# B&R Automation Studio project Myjnia
Automation Studio 4.9.3.144 SP; technology packages: mappView 5.12.1

## Configuration Config1

CPU X20CP1382, AutomationRuntime B4.83, Build 4.1.2, Vc V4.72.2

### Task classes (Cpu.sw)
```
Cyclic#4:
  Program <- Program.prg
VcDataObjects: Visu <- Visu.dob
```

### Hardware
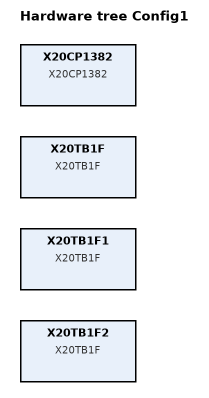
```
X20CP1382 : X20CP1382 v1.11.0.0  [X1 -> X1.SL; X2 -> X2.SL; X3 -> X3.SL]
  Module X1 (Type=X1, Virtual=true, Version=1.11.0.0)
    Connection (Connector=SS1, TargetModule=X20TB1F, TargetConnector=SS)
    Connection (Connector=SL, TargetModule=X20CP1382, TargetConnector=X1)
  Module X2 (Type=X2, Virtual=true, Version=1.11.0.0)
    Connection (Connector=SS1, TargetModule=X20TB1F1, TargetConnector=SS)
    Connection (Connector=SL, TargetModule=X20CP1382, TargetConnector=X2)
  Module X3 (Type=X3, Virtual=true, Version=1.11.0.0)
    Connection (Connector=SS1, TargetModule=X20TB1F2, TargetConnector=SS)
    Connection (Connector=SL, TargetModule=X20CP1382, TargetConnector=X3)
  Connector IF2:
    ActivateDevice = 1
    Vnc1
    VncVcObjectName1 = Visu
    VncKeyMappingFile1 = 
    VncAuthentication1 = 1
    VncPasswordViewOnly1 = v
    VncPasswordViewControl1 = c
    VncMaxConnections1 = 10
    VncRefreshRate1 = 300
  ConfigurationID = Myjnia_Config1
  Simulation = 1
X20TB1F : X20TB1F v1.0.0.0
X20TB1F1 : X20TB1F v1.0.0.0
X20TB1F2 : X20TB1F v1.0.0.0
```

## Logical view

### Program Logical/Program (IEC)

#### Types.typ
```iecst
TYPE
	KROK :
		(
		PIANA,
		WOSK,
		BLYSK,
		WODA,
		STOP
		);
END_TYPE
```

#### Variables.var
```iecst
VAR
	water_temp : INT;
	programm : INT;
	coin : USINT;
	cabin_temp : INT;
	water_heater : BOOL;
	cabin_heater : BOOL;
	water_pump : BOOL;
	TON_1 : TON;
	time : DINT;
	foam_valve : BOOL;
	wax_valve : BOOL;
	shine_valve : BOOL;
END_VAR
```

#### Main.st
```iecst
PROGRAM _INIT
	programm:=0;
END_PROGRAM

PROGRAM _CYCLIC
//time left
	time:=(TIME_TO_DINT(TON_1.PT-TON_1.ET)/1000);
	//Turning off the machine when the time is over
	IF time=0 THEN
		TON_1.IN :=FALSE;
		TON_1.PT:=T#0s;
		programm := 0;
		TON_1.IN := 0;
	END_IF;
	//Temperature control:
	IF cabin_temp<4 THEN
		cabin_heater:=TRUE;
	ELSIF cabin_temp>12 THEN
		cabin_heater:=FALSE;
	END_IF;

	CASE programm OF
		0:
			IF water_temp<4 THEN
				water_heater := TRUE;
			ELSIF water_temp>12 THEN
				water_heater := FALSE;
			END_IF;
		1,3:
			IF water_temp<32 THEN
				water_heater:=TRUE;
			ELSE water_heater:=FALSE;
			END_IF;
			TON_1.IN := TRUE;
		2,4:
			IF water_temp<20 THEN
				water_heater:=TRUE;
			ELSE water_heater:=FALSE;
			END_IF;
			TON_1.IN := TRUE;
	END_CASE
	//Coins
	CASE coin OF
		1: TON_1.PT:=TON_1.PT + T#20s;
		2: TON_1.PT:=TON_1.PT + T#40s;
		5: TON_1.PT:=TON_1.PT + T#100s;
	END_CASE;
	coin:=0;

	//Valve control
	CASE programm OF
		0:
			foam_valve:=FALSE;
			water_pump:=FALSE;
			wax_valve:=FALSE;
			shine_valve:= FALSE;
		1: 	foam_valve:=TRUE;
			water_pump:=TRUE;
			wax_valve:=FALSE;
			shine_valve:= FALSE;
		2: 	water_pump:=TRUE;
			foam_valve:=FALSE;
			wax_valve:=FALSE;
			shine_valve:= FALSE;
		3: 	wax_valve:=TRUE;
			water_pump:=TRUE;
			foam_valve:=FALSE;
			shine_valve:= FALSE;
		4: 	shine_valve:= TRUE;
			water_pump:=TRUE;
			foam_valve:=FALSE;
			wax_valve:=FALSE;
		5:	TON_1.PT := TON_1.PT-TON_1.ET;
			TON_1.IN :=FALSE;
			programm := 0;
	END_CASE;
	//Calling timer function
	TON_1();
END_PROGRAM

PROGRAM _EXIT
	(* Insert code here *)

END_PROGRAM
```

- Visualisation Logical/Visu (not shown)

Listed in the project but not available here: Logical/Global.typ, Logical/Global.var, Logical/Libraries
